TYPE XMEAS_MBS_IDX :
(
	A_FLOW			:=1,
	D_FLOW			:=2,
	E_FLOW			:=3,
	P_REACTOR		:=4,
	AC_FLOW			:=4
);
END_TYPE

(* stored: Version 1.1.0.1, ProductVersion 3.1.0.36
   DUT XMEAS_MBS_IDX: Id {ce87c558-2c19-4bb3-9db1-e0b419cf6aa1} *)
